(* IEC 61131-3 sources: Std_PalletMover/Class/HMIHandler, 1 file *)

(* ---- HMIHandler.st ---- *)
#define HMI_STATUS_OK   1
#define HMI_STATUS_WARN 2
#define HMI_STATUS_STOP 3

(*!
<Class
	Name               = "HMIHandler"
	Revision           = "0.0"
	RealtimeTask       = "false"
	CyclicTask         = "true"
	BackgroundTask     = "false"
	Sigmatek           = "false"
	OSInterface        = "false"
	HighPriority       = "false"
	Automatic          = "false"
	UpdateMode         = "Prescan"
	SharedCommandTable = "true"
	Objectsize         = "(608,120)">
	<Channels>
		<Server Name="ActiveIOObject" Visualized="true" Initialize="false" WriteProtected="false" Retentive="false"/>
		<Server Name="ClassSvr" Visualized="false" Initialize="false" WriteProtected="true" Retentive="false"/>
		<Server Name="HMIEstopStatus" Visualized="true" Initialize="false" WriteProtected="true" Retentive="false"/>
		<Server Name="HMIScanner1Status" Visualized="true" Initialize="false" WriteProtected="true" Retentive="false"/>
		<Server Name="HMIScanner2Status" Visualized="true" Initialize="false" WriteProtected="true" Retentive="false"/>
		<Server Name="HMIScanner3Status" Visualized="false" Initialize="false" WriteProtected="true" Retentive="false"/>
		<Server Name="HMIWirelessStatus" Visualized="true" Initialize="false" WriteProtected="true" Retentive="false"/>
		<Server Name="ResetToHMI" Visualized="false" Remotely="true" Initialize="false" WriteProtected="false" Retentive="false"/>
		<Client Name="MESOnline" Required="true" Internal="false"/>
		<Client Name="objStateControl" Required="true" Internal="false"/>
		<Client Name="ResetButtonHardware" Required="true" Internal="false"/>
		<Client Name="ResetButtonRemote" Required="true" Internal="false"/>
	</Channels>
</Class>
*)
HMIHandler : CLASS
	TYPE
	  eMessageResponse :  //! <Type Public="true" Name="eMessageResponse"/>
	  (
	    mr_Idle,
	    mr_Positive,
	    mr_Negative
	  )$UDINT;
#pragma pack(push, 1)
	  tHMIMessage : STRUCT  //! <Type Public="true" Name="tHMIMessage"/>
	    hm_Enable : BOOL;
	    hm_pMessage : ^CHAR;
	  END_STRUCT;
#pragma pack(pop)
#pragma pack(push, 1)
	  tHMIMessageResponse : STRUCT  //! <Type Public="true" Name="tHMIMessageResponse"/>
	    hmr_Enable : BOOL;
	    hmr_pMessage : ^CHAR;
	    hmr_Response : eMessageResponse;
	  END_STRUCT;
#pragma pack(pop)
	END_TYPE
  //Servers:
	ClassSvr 	: SvrChCmd_DINT;
	HMIScanner1Status 	: SvrCh_DINT;
	HMIScanner2Status 	: SvrCh_DINT;
	HMIScanner3Status 	: SvrCh_DINT;
	HMIEstopStatus 	: SvrCh_DINT;
	HMIWirelessStatus 	: SvrCh_DINT;
	ActiveIOObject 	: SvrCh_DINT;
	ResetToHMI 	: SvrCh_DINT;
  //Clients:
	objStateControl 	: CltChCmd_Standard;
	MESOnline 	: CltCh_DINT;
	ResetButtonRemote 	: CltCh_DINT;
	ResetButtonHardware 	: CltCh_DINT;
  //Variables:
  //Functions:

	FUNCTION VIRTUAL GLOBAL CyWork
		VAR_INPUT
			EAX 	: UDINT;
		END_VAR
		VAR_OUTPUT
			state (EAX) 	: UDINT := READY;
		END_VAR;

	FUNCTION GLOBAL GetHMIMessage
		VAR_OUTPUT
			returnValue 	: tHMIMessageResponse;
		END_VAR;

	FUNCTION GLOBAL SetHMIMessage
		VAR_INPUT
			HMIMessage 	: tHMIMessage;
		END_VAR;
  //Tables:
	FUNCTION @STD
		VAR_OUTPUT
			ret_code	: CONFSTATES;
		END_VAR;
	FUNCTION GLOBAL TAB @CT_;
END_CLASS;

#pragma usingLtd Standard

FUNCTION GLOBAL HMIHandler::GetHMIMessage
  #pragma warning(disable: 73);
  #pragma warning(disable: 76);
	VAR_OUTPUT
		returnValue 	: tHMIMessageResponse;
	END_VAR
  #pragma warning(default: 73);
  #pragma warning(default: 76);
END_FUNCTION

FUNCTION GLOBAL HMIHandler::SetHMIMessage
  #pragma warning(disable: 73);
  #pragma warning(disable: 76);
	VAR_INPUT
		HMIMessage 	: tHMIMessage;
	END_VAR
  #pragma warning(default: 73);
  #pragma warning(default: 76);
END_FUNCTION

FUNCTION VIRTUAL GLOBAL HMIHandler::CyWork
	VAR_INPUT
		EAX 	: UDINT;
	END_VAR
	VAR_OUTPUT
		state (EAX) 	: UDINT;(* := READY *)
	END_VAR
  VAR
  	tmpSafetyStatus : StateControl::tSafetyStatus;
  END_VAR

  tmpSafetyStatus := objStateControl.GetSafetyStatus();
  MESOnline := MESOnline.Read();
  ResetButtonHardware := ResetButtonHardware.Read();
  ResetButtonRemote := ResetButtonRemote.Read();

  if tmpSafetyStatus.ss_Scanner1 = StateControl::ssf_Warning then
    HMIScanner1Status := HMI_STATUS_WARN;
  elsif tmpSafetyStatus.ss_Scanner1 = StateControl::ssf_Stop | tmpSafetyStatus.ss_Scanner1 = StateControl::ssf_Estop then
    HMIScanner1Status := HMI_STATUS_STOP;
  else
    HMIScanner1Status := HMI_STATUS_OK;
  end_if;

  if tmpSafetyStatus.ss_Scanner2 = StateControl::ssf_Warning then
    HMIScanner2Status := HMI_STATUS_WARN;
  elsif tmpSafetyStatus.ss_Scanner2 = StateControl::ssf_Stop | tmpSafetyStatus.ss_Scanner2 = StateControl::ssf_Estop then
    HMIScanner2Status := HMI_STATUS_STOP;
  else
    HMIScanner2Status := HMI_STATUS_OK;
  end_if;

  if tmpSafetyStatus.ss_Estop = StateControl::es_Clear then
    HMIEstopStatus := HMI_STATUS_OK;
  elsif tmpSafetyStatus.ss_Estop = StateControl::es_PendingReset then
    HMIEstopStatus := HMI_STATUS_WARN;
  elsif tmpSafetyStatus.ss_Estop = StateControl::es_Pressed then
    HMIEstopStatus := HMI_STATUS_STOP;
  end_if;

  if MESOnline = TRUE then
    HMIWirelessStatus := HMI_STATUS_OK;
  else
    HMIWirelessStatus := HMI_STATUS_STOP;
  end_if;

  ResetToHMI := ResetButtonHardware | ResetButtonRemote;

END_FUNCTION
